TYPE ST_GCSpinAxisJogService :
STRUCT
	Ctrl : ST_GCSpinAxisJogCtrl;
	Status : ST_GCSpinAxisJogStatus;
END_STRUCT
END_TYPE

(* stored: Version 1.1.0.1, ProductVersion 3.1.4026.18
   DUT ST_GCSpinAxisJogService: Id {ec242fef-6370-456b-aa8a-3db42ab9fe47} *)
